// TIA Portal V19 export
DATA_BLOCK "Pu_GP01.GP13"   // DB1013
// stored: AutoNumber false, InstanceOfName Pu_Versorgung.GP0x, InstanceOfType FB
"Pu_Versorgung.GP0x"
   // VAR RETAIN
   //    In { ExternalVisible := 'False'; ExternalWritable := 'False'} : Struct
   //       Auto : Bool;
   //       Ein : Bool;
   //       Not_Halt : Bool;
   //       Quitt_Al_Dfl : Bool;
   //       kein_Gas_Alarm : Bool;
   //       Leckage_Pumpe_ok : Bool;
   //       Leckage_PFA_Uebergang_ok : Bool;
   //       Leckage_Doppelrohr_ok : Bool;
   //       Leckage_Uml_Tunnel_ok : Bool;
   //       Leckage_Doppelschlauch_ok : Bool;
   //       Niv_min : Bool;
   //       Niv_max : Bool;
   //       Niv_Min_CM01 : Bool;
   //       Niv_Max_CM01 : Bool;
   //       Niv_Übervoll_CM01 : Bool;
   //       Niv_Min_CM02 : Bool;
   //       Niv_Max_CM02 : Bool;
   //       Niv_Übervoll_CM02 : Bool;
   //       Frg_Niv_CM05 : Bool;
   //       SRM_Saugseite_auf : Bool;
   //       SRM_Saugseite_zu : Bool;
   //       SRM_Druckseite_auf : Bool;
   //       SRM_Druckseite_zu : Bool;
   //       SRM_Eingang_Spülltg_auf : Bool;
   //       SRM_Eingang_Spülltg_zu : Bool;
   //       SRM_Ausgang_Spülltg_auf : Bool;
   //       SRM_Ausgang_Spülltg_zu : Bool;
   //       SRM_Versogung_UV01_auf : Bool;
   //       SRM_Versogung_UV01_zu : Bool;
   //       SRM_UV01_CM01_auf : Bool;
   //       SRM_UV01_CM01_zu { ExternalAccessible := 'False'} : Bool;
   //       SRM_UV01_CM02_auf { ExternalAccessible := 'False'} : Bool;
   //       SRM_UV01_CM02_zu { ExternalAccessible := 'False'} : Bool;
   //       Anf_HF_CM01 { ExternalAccessible := 'False'} : Bool;
   //       Anf_HF_CM02 { ExternalAccessible := 'False'} : Bool;
   //       IBC_vorhanden { ExternalAccessible := 'False'} : Bool;
   //       Tuer_vorn_zu { ExternalAccessible := 'False'} : Bool;
   //       Tuer_seitlich_zu { ExternalAccessible := 'False'} : Bool;
   //       Imp_Dfl { ExternalAccessible := 'False'} : Bool;
   //       GW_Dfl { ExternalAccessible := 'False'} : Bool;
   //       Betriebsart { ExternalAccessible := 'False'} : USInt;
   //       Niveau { ExternalAccessible := 'False'} : USInt;
   //       Dfl { ExternalAccessible := 'False'} : Real;
   //    END_STRUCT;
   //    Param { ExternalAccessible := 'False'; ExternalVisible := 'False'; ExternalWritable := 'False'} : Struct
   //       Spülzeit : Time;
   //    END_STRUCT;
   //    Zst { ExternalAccessible := 'False'; ExternalVisible := 'False'; ExternalWritable := 'False'} : Struct
   //       Niveau : USInt;
   //       Status_GP0x : USInt;
   //       Restzeit_Spülen : Time;
   //       Spuelen : Bool;
   //       Pumpen : Bool;
   //       Weg_frei : Bool;
   //       Spuelen_aktiv : Bool;
   //       Bedienung_erlaubt : Bool;
   //    END_STRUCT;
   //    Mld { ExternalVisible := 'False'; ExternalWritable := 'False'} : Struct
   //       Leckage_Pumpe : Bool;
   //       Leckage_PFA_Uebergang : Bool;
   //       Leckage_Doppelrohr : Bool;
   //       Leckage_Uml_Tunnel : Bool;
   //       Leckage_Doppelschlauch : Bool;
   //       Niv_Sensorfehler : Bool;
   //       GW_Dfl : Bool;
   //       UeW_Dfl_Dos : Bool;
   //       Leermeldung : Bool;
   //       Vollmeldung : Bool;
   //       n_Auto : Bool;
   //       Radarsonde_niO : Bool;
   //    END_STRUCT;
   //    Out { ExternalVisible := 'False'; ExternalWritable := 'False'} : Struct
   //       GP0x_Ein : Bool;
   //       Spülventil_Eingang : Bool;
   //       Spülventil_Ausgang : Bool;
   //       Ventil_Saugseite : Bool;
   //       Ventil_Druckseite : Bool;
   //       Ventil_Entsorgung : Bool;
   //       Versorgung_UV01 : Bool;
   //       UV01_CM01 : Bool;
   //       UV01_CM02 : Bool;
   //    END_STRUCT;
   // END_VAR
   // VAR
   //    IEC_Timer : Struct
   //       GW_Dfl { ExternalAccessible := 'False'; ExternalVisible := 'False'; ExternalWritable := 'False'; S7_SetPoint := 'True'} : TON_TIME;
   //       Spülen { S7_SetPoint := 'True'} : TP_TIME;
   //       Verz_Min { S7_SetPoint := 'True'} : TON_TIME;
   //       Imp_Dfl { S7_SetPoint := 'True'} : TON_TIME;
   //       Spülventil_Ausgang { S7_SetPoint := 'True'} : TOF_TIME;
   //       Verz_NivMax { S7_SetPoint := 'True'} : TON_TIME;
   //    END_STRUCT;
   //    R_TRIG_Hand_EIN { S7_SetPoint := 'True'} : R_TRIG;
   // END_VAR
BEGIN
END_DATA_BLOCK
